// TIA Portal V16 export
// export: Created 2025-08-30T12:59:07.9958336Z, ExportSetting WithDefaults, DisplayName Totally Integrated Automation Portal, DisplayVersion V16, DisplayName TIA Portal Version Control Interface, DisplayVersion V16, DisplayName TIA Portal Openness, DisplayVersion V16, DisplayName STEP 7 Professional, DisplayVersion V16, DisplayName STEP 7 Safety, DisplayVersion V16, DisplayName WinCC Advanced, DisplayVersion V16
FUNCTION "SiemensEnc" : Void   // FC15, STL
TITLE = Test Siemens ENCODER
VERSION : 0.1
// stored: AutoNumber true, UDAEnableTagReadback false
BEGIN

NETWORK
TITLE = Presettings
      L     0;  //Delete control bits
      T     %DB1.DBD0;
      T     %DB1.DBD4;
      SET;
      S     %DB1.DBX4.0;  //Open SW gate









NETWORK
TITLE = Write to the control interface

NETWORK
TITLE = Read from the feedback interface
//Read 8 bytes from the 1 Count24V
//Configured start address of inputs
      L     "Tag_25":P;
      T     %DB1.DBD8;
      L     "Tag_26":P;
      T     %DB1.DBD12;
      R     %DB1.DBX4.0;  //Close SW gate



END_FUNCTION
